FUNCTION_BLOCK FB_JointBase
VAR_INPUT
END_VAR
VAR_OUTPUT
END_VAR
VAR
	// arm and joint index
	m_armIdx :INT;
	m_jntIdx :INT;
	
	// motor IO
	m_motorInputs AT%I*	:ST_MotorInputs;
	m_motorOutputs AT%Q* :ST_MotorOutputs;
	
	// cycle time
	m_cycleTime :LREAL;
	
	// calibrated link encoder data
	m_minLinkEncoder :DINT;
	m_maxLinkEncoder :DINT;
	m_caliLinkEncoder :DINT;
	m_linkEncCaliJntPos :LREAL;
	m_linkEncZeroCross :INT;
	m_initMotorEnc : DINT;
	m_multiCycles :INT;
	
	// joint position from link encoder after power on
	m_initLinkPos :LREAL;
	
	// data for link encoder multiple cycles
	m_lastLinkEncoder :DINT;
	m_linkEncCycles:INT;
	
	// device paramters
	m_motorEncoderRes :DINT;
	m_linkEncoderRes :DINT;
	m_motorReduction :LREAL;
	m_linkEncoderReduction :LREAL;
	m_trqConst :LREAL;
	m_maxCurrent :LREAL;
	m_motorDir :INT;								
	m_linkEncoderDir :INT;
	m_minJntPos: LREAL;
	m_maxJntPos: LREAL;
	
	// macro defined data for quick calculation
	m_trq2CurrentRatio:LREAL;
	m_current2TrqRatio:LREAL;
	m_linkEnc2PosRatio :LREAL;
	m_motorEnc2PosRatio :LREAL;
	
	// joint data
	m_curMotorPos :LREAL;
	m_curLinkPos :LREAL;
	m_curLinkSingle :LREAL;
	m_curJntPos	:LREAL;
	m_curJntVel :LREAL;
	m_rawJntVel :LREAL;
	m_curJntTrq :	LREAL;
	m_rawCurrent : LREAL;
	m_filtCurrent : LREAL;
	m_cmdJntPos :LREAL;
	m_cmdJntVel :LREAL;
	m_cmdJntTrq :LREAL;
	m_cmdCurrent : LREAL;
	m_lastJntPos :LREAL;
	
	// velocity filter
	m_jntVelLpf :FB_LowPassFilter;
	
	// command torque filter
	m_curTrqLpf : FB_LowPassFilter;
	m_cmdTrqLpf :FB_LowPassFilter;
	
	// velocity is calculated every (m_velCalcCycles) control cycles
	// TODO: insturment joint motor can not reach 4k now, so calculate their velocity with 1k frequency, need to remove later
	m_velCalcCycles :INT :=1;
	m_curVelCalCycles :INT :=1;
	
	// SDO writer
	m_opModeSDOWrite:FB_EcCoESdoWrite;
	m_MotorCurrentSDOWrite:FB_EcCoESdoWrite;
END_VAR

PROPERTY cmdCurrent : LREAL
GET
cmdCurrent:=m_cmdCurrent;
END_GET
END_PROPERTY

METHOD PUBLIC disable : BOOL
VAR_INPUT
END_VAR
m_motorOutputs.m_controlWord:=DriverCtrlWord_INIT;
disable:=true;
END_METHOD

METHOD PUBLIC enable : BOOL
VAR_INPUT
END_VAR
IF DriverStatusWord_INIT = m_motorInputs.m_statusWord THEN
	m_motorOutputs.m_controlWord:=DriverCtrlWord_PREOP;
	enable := FALSE;
ELSIF DriverStatusWord_PREOP = m_motorInputs.m_statusWord THEN
	m_motorOutputs.m_controlWord:=DriverCtrlWord_OP;
	enable :=  FALSE;
ELSIF DriverStatusWord_OP = m_motorInputs.m_statusWord THEN
	enable :=  TRUE;
//ELSE
//	m_motorOutputs.m_controlWord:=DriverCtrlWord_INIT;
//	enable :=  FALSE;
END_IF
END_METHOD

PROPERTY filtCurrent : LREAL
GET
filtCurrent:=m_filtCurrent;
END_GET
END_PROPERTY

METHOD initJntPos : BOOL
VAR_INPUT
END_VAR
m_lastLinkEncoder :=m_motorInputs.m_linkEncoder;
m_linkEncCycles:=0;
m_curLinkPos :=linkEnc2Pos();
m_initLinkPos:=m_curLinkPos;
m_initMotorEnc :=m_motorInputs.m_motorEncoder;
m_curMotorPos:=motorEnc2Pos();
m_curJntPos := m_curMotorPos;
m_cmdJntPos :=m_curJntPos;	
m_lastJntPos :=m_curJntPos;
END_METHOD

PROPERTY initLinkPos : lreal
GET
initLinkPos:=m_initLinkPos;
END_GET
SET
m_initLinkPos:=initLinkPos;
END_SET
END_PROPERTY

METHOD isEnabled : BOOL
VAR_INPUT
END_VAR
isEnabled :=(DriverStatusWord_OP = m_motorInputs.m_statusWord);
END_METHOD

PROPERTY jntPos : LREAL
GET
jntPos := m_curJntPos;
END_GET
END_PROPERTY

PROPERTY jntTrq : LREAL
GET
jntTrq:=m_curJntTrq;
END_GET
END_PROPERTY

PROPERTY jntVel : LREAL
GET
jntVel := m_curJntVel;
END_GET
END_PROPERTY

METHOD PROTECTED linkEnc2Pos : LREAL
VAR_INPUT
END_VAR
VAR
	incLinkPos :LREAL;
	newLinkEnc :DINT;
END_VAR
// cycle check
IF 1=m_multiCycles THEN
	IF (m_motorInputs.m_linkEncoder - m_lastLinkEncoder)*m_linkEncoderDir < -m_linkEncoderRes/2 THEN
		m_linkEncCycles :=m_linkEncCycles+1;
	ELSIF (m_motorInputs.m_linkEncoder - m_lastLinkEncoder)*m_linkEncoderDir > m_linkEncoderRes/2 THEN
		m_linkEncCycles :=m_linkEncCycles-1;
	END_IF
END_IF
m_lastLinkEncoder:=m_motorInputs.m_linkEncoder;

// convert link encoder if joint cross zero
newLinkEnc := m_motorInputs.m_linkEncoder;
IF 1=m_linkEncZeroCross AND 0 = m_multiCycles THEN
	IF 1=m_linkEncoderDir AND m_motorInputs.m_linkEncoder < m_minLinkEncoder THEN
		newLinkEnc := m_motorInputs.m_linkEncoder + m_linkEncoderRes;
	ELSIF -1=m_linkEncoderDir AND m_motorInputs.m_linkEncoder < m_maxLinkEncoder THEN
		newLinkEnc := m_motorInputs.m_linkEncoder + m_linkEncoderRes;
	END_IF
END_IF

// motion from calibrated points
incLinkPos := (newLinkEnc-m_caliLinkEncoder)*m_linkEnc2PosRatio;

// absolute joint position
linkEnc2Pos := incLinkPos + m_linkEncCaliJntPos + 2*PI* m_linkEncCycles;
END_METHOD

METHOD linkEnc2Single : LREAL
VAR_INPUT
END_VAR
linkEnc2Single := m_motorInputs.m_linkEncoder*m_linkEnc2PosRatio;
END_METHOD

PROPERTY PUBLIC linkPos : LREAL
GET
linkPos:=m_curLinkPos;
END_GET
END_PROPERTY

PROPERTY linkSingle : LREAL
GET
linkSingle :=m_curLinkSingle;
END_GET
END_PROPERTY

METHOD PUBLIC motorEnc2Pos : LREAL
VAR_INPUT
END_VAR
motorEnc2Pos:= (m_motorInputs.m_motorEncoder-m_initMotorEnc)* m_motorEnc2PosRatio +m_initLinkPos;
END_METHOD

PROPERTY PUBLIC motorPos : LREAL
GET
motorPos := m_curMotorPos;
END_GET
END_PROPERTY

METHOD PROTECTED motorPos2Enc : DINT
VAR_INPUT
	i_jntPos :LREAL;
END_VAR

VAR
END_VAR
motorPos2Enc := LREAL_TO_DINT((i_jntPos-m_initLinkPos)/m_motorEnc2PosRatio + m_initMotorEnc);
END_METHOD

PROPERTY rawCurrent : LREAL
GET
rawCurrent := m_rawCurrent;
END_GET
END_PROPERTY

METHOD PUBLIC updateCmds : BOOL
VAR_INPUT
	i_opMode : E_DriverOPMode;
	i_cmdPos :LREAL;
	i_cmdTrq :LREAL;
END_VAR
VAR
	filtCmdTrq :LREAL;
END_VAR
m_motorOutputs.m_opMode:=INT_TO_SINT( i_opMode);
// pos mode
IF i_opMode = DriverOPMode_Pos THEN
	m_motorOutputs.m_cmdCurrent:=0;
	m_cmdTrqLpf.reset();	
//	i_cmdPos:=LIMIT(m_minJntPos, i_cmdPos, m_maxJntPos); // May cause position jump, Do this in safety check. 
	m_cmdJntPos :=i_cmdPos;
	m_motorOutputs.m_cmdMotorEncoder :=motorPos2Enc(m_cmdJntPos);
ELSIF i_opMode = DriverOPMode_Trq THEN
	filtCmdTrq:=m_cmdTrqLpf.run(i_cmdTrq);
	m_motorOutputs.m_cmdCurrent:=LREAL_TO_DINT(LIMIT(-m_maxCurrent, filtCmdTrq*m_trq2CurrentRatio,m_maxCurrent));
	m_motorOutputs.m_cmdMotorEncoder :=m_motorInputs.m_motorEncoder; 
END_IF
m_cmdCurrent:=m_motorOutputs.m_cmdCurrent;
END_METHOD

METHOD PUBLIC updateStatus : BOOL
VAR_INPUT
END_VAR
// compute joint position
m_curLinkPos:= linkEnc2Pos();
//m_curLinkSingle:= linkEnc2Single();
m_curMotorPos:=motorEnc2Pos();
m_curJntPos := m_curMotorPos;
m_curLinkSingle := m_curLinkPos - 2*PI* m_linkEncCycles;

// compute joint velocity
m_curVelCalCycles := m_curVelCalCycles+1;
IF m_curVelCalCycles > m_velCalcCycles THEN
	m_rawJntVel:= (m_curJntPos-m_lastJntPos)/(m_cycleTime*m_velCalcCycles);
	m_curJntVel := m_jntVelLpf.run(m_rawJntVel);
	m_lastJntPos :=m_curJntPos;	
	m_curVelCalCycles:=1;
END_IF


// current and torque
m_rawCurrent := m_motorInputs.m_current;
m_filtCurrent := m_curTrqLpf.run(m_rawCurrent);
m_curJntTrq := m_filtCurrent * m_current2TrqRatio;
END_METHOD

END_FUNCTION_BLOCK

(* stored: Version 1.1.0.1, ProductVersion 3.1.4024.11
   POU FB_JointBase: Id {9ce08388-a134-4497-8af1-f051329728ca}, SpecialFunc None
   Folder property: Id {cdcb62c8-2a8b-4700-ad38-db65527ef407}
   Property cmdCurrent: Id {f0454860-a96c-4f8b-8a2f-46843af60044}
   Get Get: Id {e9954b3f-6116-4864-8a9d-3960b55dc914}
   Method disable: Id {e31df8a7-8ce0-47c3-be01-feb458684c41}
   Method enable: Id {cf1e8549-8fbc-49c1-a41e-ead1f2db1255}
   Property filtCurrent: Id {311cc4f0-6471-4110-900a-4f36251b16c7}
   Get Get: Id {48a0d0d5-f074-4a51-82e8-46c72739adae}
   Method initJntPos: Id {c1110436-e250-45fb-8008-63b89ff1e4a3}
   Property initLinkPos: Id {d7776925-1122-4a68-9f90-f18c7af4e629}
   Get Get: Id {d7e38c99-fc3b-4588-a2f6-017421dc91a7}
   Set Set: Id {36303120-5670-4aa9-aa7e-461e087d0eb8}
   Method isEnabled: Id {6575d317-fe99-4038-982b-c3651c898873}
   Property jntPos: Id {7c60c4ea-0665-427c-81ff-ecca027383e5}
   Get Get: Id {0999bfb4-2d73-48db-9f0b-eb60a7757215}
   Property jntTrq: Id {24f2edfa-7ea0-460c-b46c-37e80340999b}
   Get Get: Id {a73a2159-96f0-4307-8408-692459f39004}
   Property jntVel: Id {9f6c9647-33be-4e59-a761-fc40f97a604f}
   Get Get: Id {dda73f9b-c1f5-4fa7-a73f-7b4550e82f69}
   Method linkEnc2Pos: Id {ee202f01-7eae-4c96-9148-de033a227f8f}
   Method linkEnc2Single: Id {c72ce21a-90a5-4620-9422-56ee841650c3}
   Property linkPos: Id {e503da77-c373-4ba2-b314-228646ff52c0}
   Get Get: Id {057e650e-064f-4e5d-ae71-67363977daff}
   Property linkSingle: Id {155bff3b-1577-4b32-ab22-9100cfe6ef2e}
   Get Get: Id {fd091afb-c96c-47ba-b624-538017ea6b03}
   Method motorEnc2Pos: Id {5111dbab-73a3-4041-b0b2-3d1b70394152}
   Property motorPos: Id {257e5d05-bbd2-45b4-a27c-60112e2ac416}
   Get Get: Id {5c2a1542-7420-4542-ba4a-8202be5bc4e5}
   Method motorPos2Enc: Id {5927a17d-d8e9-40fc-9c34-e6793775a7fc}
   Property rawCurrent: Id {29700c1a-0c89-4de7-9040-f5ad478f605c}
   Get Get: Id {efca7981-2ed8-4e66-9338-eb89f6555374}
   Method updateCmds: Id {a4f5fe94-40e9-4f77-a4d8-a2af848a52e6}
   Method updateStatus: Id {77cc6f91-59d3-42a9-8d8a-2f8d584653fb} *)
